FUNCTION_BLOCK FB_HwTrayLockControl
VAR_INPUT
	bExecute		: BOOL;
	eCtrl			: E_LockCtrl;
END_VAR
VAR_OUTPUT
	bBusy 		: BOOL;
	bError 		: BOOL;
	nErrorId	: ERRORID;	
END_VAR
VAR_IN_OUT
	pHwRef : POINTER TO FB_HwRefTrayLock;
END_VAR
VAR
	nState		: USINT;
	timer		: TON;
END_VAR

IF bExecute THEN
	IF pHwRef = 0 THEN
		bError := TRUE;
		nErrorId := E_ErrorIdHwGeneral.ERRORID_InvalidHwRef;
		RETURN;
	END_IF

	CASE nState OF
		0:	IF eCtrl = E_LockCtrl.Unlock THEN
				IF pHwRef^.eCurrentState = E_LockState.Unlocked THEN
					RETURN;
				ELSE
					bBusy := TRUE;
					nState := 1; //Unlocking
				END_IF
			ELSE
				IF pHwRef^.eCurrentState = E_LockState.Locked THEN
					RETURN;
				ELSE
					bBusy := TRUE;
					nState := 10; //Locking
				END_IF
			END_IF
			
		1:	//Unlocking, disable heater
			pHwRef^.bDisableHeater := TRUE;
			timer(IN:= TRUE, PT:= T#200MS);
			nState := 2;
			
		2:	//Time elapsed?
			timer();
			IF timer.Q THEN
				timer(IN:= FALSE);
				nState := 3;
			END_IF
			
		3:	//Set outputs
			pHwRef^.bLock := FALSE;
			pHwRef^.bUnlock := TRUE;
			timer(IN:= TRUE, PT:= T#3S); //Timeout
			IF pHwRef^.P_bFeedback THEN
				IF pHwRef^.bUnlocked THEN
					nState := 80;
				ELSIF timer.Q THEN
					nErrorId := E_ErrorIdHwGeneral.ERRORID_UnlockingFailed;
					nState := 99; //Error
				END_IF
			ELSE
				IF timer.Q THEN
					nState := 80;
				END_IF
			END_IF
			
		10: //Locking
			pHwRef^.bLock := TRUE;
			pHwRef^.bUnlock := FALSE;
			timer(IN:= TRUE, PT:= T#3S); //Timeout
			IF pHwRef^.P_bFeedback THEN
				IF pHwRef^.bLocked THEN
					//Enable heater
					pHwRef^.bDisableHeater := FALSE;
					nState := 80;
				ELSIF timer.Q THEN
					nErrorId := E_ErrorIdHwGeneral.ERRORID_LockingFailed;
					nState := 99; //Error
				END_IF
			ELSE
				IF timer.Q THEN
					nState := 80;
				END_IF
			END_IF
	END_CASE
	
	IF nState >= 80 THEN
		pHwRef^.bLock := FALSE;
		pHwRef^.bUnlock := FALSE;
		bBusy := FALSE;
		IF nState = 99 THEN
			bError := TRUE;
		END_IF
	END_IF

ELSE
	timer(IN:= FALSE);
	bBusy := FALSE;
	bError := FALSE;
	nErrorId := 0;
	nState := 0;	
END_IF

END_FUNCTION_BLOCK

(* stored: Version 1.1.0.1, ProductVersion 3.1.4024.11
   POU FB_HwTrayLockControl: Id {2d2ea207-d808-444d-8a0d-7ebcc53e7717}, SpecialFunc None *)
